# EPICS substitutions: iocs/testSmaract/testSmaractApp/Db/testSmaract_expanded.substitutions
# This file was automatically generated on Fri 13 May 2016 13:02:24 BST from
# source: /home/hgv27681/R3.14.12.3/support/smaractEcm/etc/makeIocs/testSmaract.xml
#
# *** Please do not edit this file: edit the source file instead. ***
#

# Macros:
#  P        EPICS name prefix
#  R        EPICS name suffix
#  PORT     Asyn port
#  TIMEOUT  Timeout
file $(SMARACTECM)/db/smaractEcmController.template
{
pattern { P, R, PORT, TIMEOUT }
    { "TEST-MO-SPOD-01", "ECM1", "ecm1", "0" }
}

# Macros:
#  name  axis name
file $(SMARACTECM)/db/smarpodAxis.template
{
pattern { P, R, PORT, AXIS, TIMEOUT, name }
    { "TEST-MO-SPOD-01:A", "X", "ecm1", "1", "1", "AX" }
    { "TEST-MO-SPOD-01:A", "Y", "ecm1", "2", "1", "AY" }
    { "TEST-MO-SPOD-01:A", "Z", "ecm1", "3", "1", "AZ" }
    { "TEST-MO-SPOD-01:A", "RX", "ecm1", "4", "1", "ARX" }
    { "TEST-MO-SPOD-01:A", "RY", "ecm1", "5", "1", "ARY" }
    { "TEST-MO-SPOD-01:A", "RZ", "ecm1", "6", "1", "ARZ" }
}

# Macros:
#  P           Device Prefix
#  M           Device Suffix
#  PORT        Asyn port for motor record
#  ADDR        Address on controller
#  DESC        Description, displayed on EDM screen
#  MRES        Motor Step Size (EGU)
#  VELO        Velocity (EGU/s)
#  PREC        Display Precision
#  EGU         Engineering Units
#  TWV         Tweak Step Size (EGU)
#  DTYP        DTYP of record
#  DIR         User Direction
#  VBAS        Base Velocity (EGU/s)
#  VMAX        Max Velocity (EGU/s), defaults to VELO
#  ACCL        Seconds to Velocity
#  BDST        BL Distance (EGU)
#  BVEL        BL Velocity (EGU/s)
#  BACC        BL Seconds to Veloc.
#  DHLM        Dial High Limit
#  DLLM        Dial Low Limit
#  HLM         User High Limit
#  LLM         User Low Limit
#  HLSV        HW Lim. Violation Svr
#  INIT        Startup commands
#  SREV        Steps per Revolution
#  RRES        Readback Step Size (EGU)
#  ERES        Encoder Step Size (EGU)
#  JAR         Jog Acceleration (EGU/s^2)
#  UEIP        Use Encoder If Present
#  URIP        Use RDBL If Present
#  RDBL        Readback Location, set URIP = 1 if you specify this
#  RTRY        Max retry count
#  DLY         Readback settle time (s)
#  OFF         User Offset (EGU)
#  RDBD        Retry Deadband (EGU)
#  FOFF        Freeze Offset, 0=variable, 1=frozen
#  ADEL        Alarm monitor deadband (EGU)
#  NTM         New Target Monitor, only set to 0 for soft motors
#  FEHIGH      HIGH limit for following error
#  FEHIHI      HIHI limit for following error
#  FEHHSV      HIHI alarm severity for following error
#  FEHSV       HIGH alarm severity for following error
#  SCALE       Scale factor, if pmacSetAxisScale is used this should be set
#  HOMEVIS     If 1 then home is visible on the gui
#  HOMEVISSTR  If HOMEVIS=0, then display this text on the gui instead
#  name        Object name and gui association name
#  alh         Set this to alh to add the motor to the alarm handler and send emails,
#  gda_name    Name to export this as to GDA
#  gda_desc    Description to export this as to GDA
file $(MOTOR)/db/basic_asyn_motor.template
{
pattern { P, M, PORT, ADDR, DESC, MRES, VELO, PREC, EGU, TWV, DTYP, DIR, VBAS, VMAX, ACCL, BDST, BVEL, BACC, DHLM, DLLM, HLM, LLM, HLSV, INIT, SREV, RRES, ERES, JAR, UEIP, URIP, RDBL, RTRY, DLY, OFF, RDBD, FOFF, ADEL, NTM, FEHIGH, FEHIHI, FEHHSV, FEHSV, SCALE, HOMEVIS, HOMEVISSTR, name, alh, gda_name, gda_desc }
    { "TEST-MO-SPOD-01", "X", "<iocbuilder.modules.smaractEcm.SmaractEcmController object at 0x1620050>", "1", "X Translation", "0.001", "50", "3", "um", "1000", "asynMotor", "0", "0", "$(VELO)", "0.5", "0", "0", "", "8000", "-8000", "", "", "MAJOR", "", "200", "", "0.001", "", "0", "0", "", "0", "0", "0", "", "0", "0", "1", "0", "0", "NO_ALARM", "NO_ALARM", "1", "1", "Use motor summary screen", "X", "None", "X", "$(DESC)" }
    { "TEST-MO-SPOD-01", "Y", "<iocbuilder.modules.smaractEcm.SmaractEcmController object at 0x1620050>", "2", "Y Translation", "0.001", "50", "3", "um", "1000", "asynMotor", "0", "0", "$(VELO)", "0.5", "0", "0", "", "8000", "-8000", "", "", "MAJOR", "", "200", "", "0.001", "", "0", "0", "", "0", "0", "0", "", "0", "0", "1", "0", "0", "NO_ALARM", "NO_ALARM", "1", "1", "Use motor summary screen", "Y", "None", "Y", "$(DESC)" }
    { "TEST-MO-SPOD-01", "Z", "<iocbuilder.modules.smaractEcm.SmaractEcmController object at 0x1620050>", "3", "Z Translation", "0.001", "50", "3", "um", "1000", "asynMotor", "0", "0", "$(VELO)", "0.5", "0", "0", "", "8000", "-8000", "", "", "MAJOR", "", "200", "", "0.001", "", "0", "0", "", "0", "0", "0", "", "0", "0", "1", "0", "0", "NO_ALARM", "NO_ALARM", "1", "1", "Use motor summary screen", "Z", "None", "Z", "$(DESC)" }
    { "TEST-MO-SPOD-01", "RX", "<iocbuilder.modules.smaractEcm.SmaractEcmController object at 0x1620050>", "4", "X Rotation", "0.001", "10", "3", "udeg", "1000", "asynMotor", "0", "0", "$(VELO)", "0.5", "0", "0", "", "8000", "-8000", "", "", "MAJOR", "", "200", "", "0.001", "", "0", "0", "", "0", "0", "0", "", "0", "0", "1", "0", "0", "NO_ALARM", "NO_ALARM", "1", "1", "Use motor summary screen", "RX", "None", "RX", "$(DESC)" }
    { "TEST-MO-SPOD-01", "RY", "<iocbuilder.modules.smaractEcm.SmaractEcmController object at 0x1620050>", "5", "Y Rotation", "0.001", "10", "3", "udeg", "1000", "asynMotor", "0", "0", "$(VELO)", "0.5", "0", "0", "", "8000", "-8000", "", "", "MAJOR", "", "200", "", "0.001", "", "0", "0", "", "0", "0", "0", "", "0", "0", "1", "0", "0", "NO_ALARM", "NO_ALARM", "1", "1", "Use motor summary screen", "RY", "None", "RY", "$(DESC)" }
    { "TEST-MO-SPOD-01", "RZ", "<iocbuilder.modules.smaractEcm.SmaractEcmController object at 0x1620050>", "6", "Z Rotation", "0.001", "10", "3", "udeg", "1000", "asynMotor", "0", "0", "$(VELO)", "0.5", "0", "0", "", "8000", "-8000", "", "", "MAJOR", "", "200", "", "0.001", "", "0", "0", "", "0", "0", "0", "", "0", "0", "1", "0", "0", "NO_ALARM", "NO_ALARM", "1", "1", "Use motor summary screen", "RZ", "None", "RZ", "$(DESC)" }
}
